{attribute 'qualified_only'}
{attribute 'strict'}
TYPE EReportType_t :
(
	eCoverageReport := 1,
	eUnitTestReport := 2,
	eExternalReport
);
END_TYPE

(* stored: Version 1.1.0.1, ProductVersion 3.1.4024.3
   DUT EReportType_t: Id {ab003a45-b18c-4681-8257-cc03762f6df4} *)
